# B&R Automation Studio project RunninLights
Automation Studio 4.3.3.196

## Configuration Config1

CPU X20CP1382, AutomationRuntime I4.33, Build 4.1.2, Vc V4.33.0

### Task classes (Cpu.sw)
```
Cyclic#4:
  RunningLig <- RunningLights.prg
  DrawingRob <- DrawingRobot.prg
VcDataObjects: Visual <- VisualSDU.dob
Libraries: standard
```

### Hardware
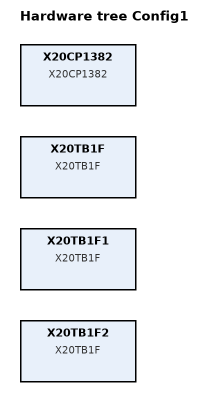
```
X20CP1382 : X20CP1382 v1.3.2.0  [X1 -> X1.SL; X2 -> X2.SL; X3 -> X3.SL]
  Module X1 (Type=X1, Virtual=true, Version=1.3.2.0)
    Connection (Connector=SS1, TargetModule=X20TB1F, TargetConnector=SS)
    Connection (Connector=SL, TargetModule=X20CP1382, TargetConnector=X1)
  Module X2 (Type=X2, Virtual=true, Version=1.3.2.0)
    Connection (Connector=SS1, TargetModule=X20TB1F1, TargetConnector=SS)
    Connection (Connector=SL, TargetModule=X20CP1382, TargetConnector=X2)
  Module X3 (Type=X3, Virtual=true, Version=1.3.2.0)
    Connection (Connector=SS1, TargetModule=X20TB1F2, TargetConnector=SS)
    Connection (Connector=SL, TargetModule=X20CP1382, TargetConnector=X3)
  Connector IF2:
    ActivateDevice = 1
    HostName = localhost
    Vnc1
    VncVcObjectName1 = Visual
    VncKeyMappingFile1 = VC\PS2-Keyboard.dis
    VncAuthentication1 = 1
    VncPasswordViewOnly1 = v
    VncPasswordViewControl1 = c
    VncRefreshRate1 = 100
  ConfigurationID = RunninLights_Config1
X20TB1F : X20TB1F v1.0.0.0
X20TB1F1 : X20TB1F v1.0.0.0
X20TB1F2 : X20TB1F v1.0.0.0
```

## Logical view

Binary libraries used (declarations not repeated): operator, runtime, astime, AsIecCon, standard


### Program Logical/RunningLights (IEC)

#### Main.st - Init, cyclic, exit code
```iecst
PROGRAM _INIT
	input := 'N1N2N3N4N5N6N7N8N7N6N5N4N3N2N1FN1N2KKKKKKN3N4N5N6N7N8Q';
	//N + tal = tænd lys #
	//K = behold gammel værdi
	//F = OFF
	//Q = Quit
END_PROGRAM

PROGRAM _CYCLIC

	timer.IN := TRUE;
	timer.PT := T#1000ms;

	IF timer.Q THEN
		i := i + 1;
		tempText := USINT_TO_STRING(i);
		visualTextCounter := 'i = 000';
		visualTextCounter := REPLACE(visualTextCounter, tempText, LEN(tempText), LEN(visualTextCounter)-LEN(tempText)+1);

		IF i < LEN(input) THEN

			commandText := MID(input, 1, i);

			IF MID(input, 1, i) = 'N' THEN
				i := i + 1;
				visualLight0 := 0;
				visualLight1 := 0;
				visualLight2 := 0;
				visualLight3 := 0;
				visualLight4 := 0;
				visualLight5 := 0;
				visualLight6 := 0;
				visualLight7 := 0;

				CASE STRING_TO_USINT(MID(input, 1, i)) OF
					1 :
						visualLight0 := 1;
					2 :
						visualLight1 := 1;
					3 :
						visualLight2 := 1;
					4 :
						visualLight3 := 1;
					5 :
						visualLight4 := 1;
					6 :
						visualLight5 := 1;
					7 :
						visualLight6 := 1;
					8 :
						visualLight7 := 1;b

				END_CASE

			ELSIF(MID(input, i, l ) = 'K') THEN
				//Keep old values
			ELSIF(MID(input, i, 1 ) = 'Q') THEN
				//Quit
				i := 0;
			ELSIF(MID(input, i, 1 ) = 'F') THEN
				visualLight0 := 0;
				visualLight1 := 0;
				visualLight2 := 0;
				visualLight3 := 0;
				visualLight4 := 0;
				visualLight5 := 0;
				visualLight6 := 0;
				visualLight7 := 0;
			END_IF

		END_IF

		timer.IN := FALSE;

	END_IF

	//Calling timer function block
	timer();

END_PROGRAM

PROGRAM _EXIT

END_PROGRAM
```

#### Variables.var - Local variables
```iecst
VAR
	timer : TON;
	i : USINT;
	tempText : STRING[20];
	visualTextCounter : STRING[20];
	visualLight1 : USINT;
	visualLight2 : USINT;
	visualLight3 : USINT;
	visualLight4 : USINT;
	visualLight5 : USINT;
	visualLight6 : USINT;
	visualLight7 : USINT;
	visualLight0 : USINT;
	commandText : STRING[10];
	input : STRING[100];
END_VAR
```

- Visualisation Logical/VisualSDU (not shown)

### Program Logical/DrawingRobot (IEC)

#### Variables.var
```iecst
VAR
	timer : TON;
	commandText : STRING[5];
	input : STRING[40000];
	test : USINT;
	i : USINT;
	STEP1 : BOOL;
	STEP2 : BOOL;
	STEP3 : BOOL;
	DIR1 : BOOL;
	DIR2 : BOOL;
	DIR3 : BOOL;
	EN1 : BOOL;
	EN2 : BOOL;
	EN3 : BOOL;
	timerSharpener : TON;
END_VAR
```

#### Main.st
```iecst
PROGRAM _INIT
	input := 'MDUMMMMMDUMMMMMDUMDUMDUMDUMDUMMMMM'
	//M = Move
	//D = Down
	//U = Up
	//N = New line
END_PROGRAM

PROGRAM _CYCLIC

	timer.IN := TRUE;
	timer.PT := T#1000ms

	IF timer.Q THEN
		i := i + 1;

		IF i < LEN(input) THEN
			//Change commandText to show the current function
			commandText := MID(input, 1, i);

			IF MID(input, 1, i) = 'M' THEN
				test := 1;
				//Code to move
			ELSIF(MID(input, 1, i) = 'D' THEN
				test := 2;
				//Code to make the robot move down
			ELSIF(MID(input, 1, i) = 'U' THEN
				test := 3;
				//Code to make the robot move up
			ELSIF(MID(input, 1, i) = 'N' THEN
				test := 4;
				//Code to make the robot go to the next line

			END_IF
		END_IF

	//Calling timer function block
	timer();

END_PROGRAM

PROGRAM _EXIT

END_PROGRAM
```

Listed in the project but not available here: Logical/Global.typ, Logical/Global.var, Logical/RunningLights/Types.typ
